FUNCTION f_Setbit64 : LWORD
VAR_INPUT
	inVal		: LWORD;
	bitNo		: DINT;
END_VAR
VAR
	wConst	: LWORD := 1;
END_VAR

f_Setbit64 := inVal OR SHL( wConst,bitNo MOD 64 );

END_FUNCTION

(* stored: Version 1.1.0.1, ProductVersion 3.1.4024.9
   POU f_Setbit64: Id {d63ae735-a42c-4737-b260-8c80cdaa858c}, SpecialFunc None *)
